FUNCTION F_PosOverLowerBound : BOOL
VAR_INPUT
    fPosition: LREAL;
    stPositionState: ST_PositionState;
END_VAR


F_PosOverLowerBound := fPosition > (stPositionState.fPosition - ABS(stPositionState.fDelta));

END_FUNCTION

(* stored: Version 1.1.0.1
   POU F_PosOverLowerBound: Id {0f84a03e-89d5-4ac7-905a-0b4508a08a18}, SpecialFunc None *)
